Staubli VAL3: onF3Event.pgx

program onF3Event()
  local string l_sEmpty
begin
  // look if the bButton is enable
  if bButton[2]
    // load the page Pallet
    l_sEmpty=""
    call loadPage("trajectory/PALLET/page_viewPallet",l_sEmpty)
  endIf
end
